PROGRAM MAIN
VAR
	
	Call_Fb_Idb: Call_Fb;
	Fixture_Idb: Clamping;
END_VAR

Call_Fb_Idb();

Fixture_Idb();

END_PROGRAM

(* stored: Version 1.1.0.1, ProductVersion 3.1.4024.16
   POU MAIN: Id {06cb9cdf-00f4-4974-bbbc-0941b7f466e4}, SpecialFunc None *)
